{attribute 'qualified_only'}
VAR_GLOBAL	
	extrusionWeight : REAL;
	
	extrusionHeight : REAL;
	extrusionWidth : REAL;
END_VAR

(* stored: Version 1.1.0.1, ProductVersion 3.1.4024.11
   GVL ExtrusionData: Id {77d6ed1f-6983-4e54-b69c-bfdffcab0faf} *)
